// TIA Portal V18 export
// export: Created 2025-12-01T17:53:14.513581Z, ExportSetting None, DisplayName Totally Integrated Automation Portal, DisplayVersion V18 Update 5, DisplayName TIA Portal Openness, DisplayVersion V18 Update 5, DisplayName TIA Portal Teamcenter Gateway, DisplayVersion V18, DisplayName TIA Portal Version Control Interface, DisplayVersion V18, DisplayName STEP 7 Professional, DisplayVersion V18 Update 5, DisplayName STEP 7 Safety, DisplayVersion V18, DisplayName WinCC Professional, DisplayVersion V18 Update 5
Screen "400Main"  1280x800, Number=400, Template=04Information
  ScreenLayer "Layer_0"
    Button "按钮_4" at 160,183 size 200x100  PictureOff=向右箭头_0, StyleItem=BtnNormal20, TextOff="产品计数 / Product Count / Výrobok Počítať"
    Button "按钮_6" at 408,183 size 200x100  PictureOff=向右箭头_0, StyleItem=BtnNormal20, TextOff="循环时间 / Cycle Time / Cyklus Čas"
